// TIA Portal V17 export
// export: Created 2025-03-05T08:02:39.5245744Z, ExportSetting WithDefaults, DisplayName Totally Integrated Automation Portal, DisplayVersion V17 Update 8, DisplayName TIA Portal Openness, DisplayVersion V17 Update 8, DisplayName TIA Portal Version Control Interface, DisplayVersion V17, DisplayName SINAMICS Startdrive Advanced, DisplayVersion V17 SP2, DisplayName SINAMICS Startdrive G110M, G120, G120C, G120D, G120P, G115D, DisplayVersion V17 SP2, DisplayName SINAMICS Startdrive G130, G150, S120, S150, SINAMICS MV, S210, DisplayVersion V17 SP2, DisplayName STEP 7 Professional, DisplayVersion V17 Update 8, DisplayName SINUMERIK ONE STEP 7 Toolbox, DisplayVersion V17 Update 12, DisplayName SINUMERIK 840D sl STEP 7 Toolbox, DisplayVersion V17 Update 12, DisplayName STEP 7 Safety, DisplayVersion V17 Update 6, DisplayName WinCC Advanced, DisplayVersion V17 Update 8
ORGANIZATION_BLOCK "OB100_RESTART"   // OB100, LAD, Startup
TITLE = "Complete Restart"
{ S7_Optimized_Access := 'FALSE' }
AUTHOR : ETXETAR
VERSION : 1.0
// stored: AutoNumber false, IsIECCheckEnabled false, SetENOAutomatically false
   VAR_TEMP
      OB100_EV_CLASS : Byte;
      OB100_STRTUP : Byte;
      OB100_PRIORITY : Byte;
      OB100_OB_NUMBR : Byte;
      OB100_RESERVED_1 : Byte;
      OB100_RESERVED_2 : Byte;
      OB100_STOP : Word;
      OB100_RESERVED_3 : Word;
      OB100_RESERVED_4 : Word;
      OB100_DATE_TIME : Date_And_Time;
      __PlcmigTempFillBits_20B0 : Array[0..7] of Bool;
   END_VAR
BEGIN

REGION Network 1: M_ONE / ESTABLISH "LOGIC 1" BIT
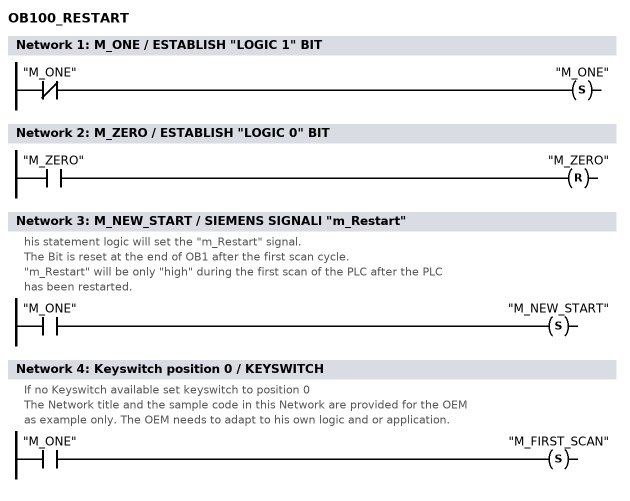
   RUNG wire#powerrail
      I_Contact( "M_ONE" )
      S_Coil( "M_ONE" )
   END_RUNG
   // the same network as SCL:
   IF NOT "M_ONE" THEN "M_ONE" := TRUE; END_IF;
END_REGION

REGION Network 2: M_ZERO / ESTABLISH "LOGIC 0" BIT
   RUNG wire#powerrail
      Contact( "M_ZERO" )
      R_Coil( "M_ZERO" )
   END_RUNG
   // the same network as SCL:
   IF "M_ZERO" THEN "M_ZERO" := FALSE; END_IF;
END_REGION

REGION Network 3: M_NEW_START / SIEMENS SIGNALl "m_Restart"
   // his statement logic will set the "m_Restart" signal.
   // The Bit is reset at the end of OB1 after the first scan cycle.
   // 
   // "m_Restart" will be only "high" during the first scan of the PLC after the PLC 
   // has been restarted.
   RUNG wire#powerrail
      Contact( "M_ONE" )
      S_Coil( "M_NEW_START" )
   END_RUNG
   // the same network as SCL:
   IF "M_ONE" THEN "M_NEW_START" := TRUE; END_IF;
END_REGION

REGION Network 4: Keyswitch position 0 / KEYSWITCH
   // If no Keyswitch available set keyswitch to position 0
   // 
   // The Network title and the sample code in this Network are provided for the OEM 
   // as example only. The OEM needs to adapt to his own logic and or application.
   RUNG wire#powerrail
      Contact( "M_ONE" )
      S_Coil( "M_FIRST_SCAN" )
   END_RUNG
   // the same network as SCL:
   IF "M_ONE" THEN "M_FIRST_SCAN" := TRUE; END_IF;
END_REGION
END_ORGANIZATION_BLOCK
